PROGRAM MAIN
VAR
	EtapeEnCours:string(50);
END_VAR
VAR // added by the converter: edge detectors and wires of the graphical bodies
    _w1, _w3, _w4, _w5, _w6, _w7, _w8, _w10 : ANY;
    _w2, _w9 : BOOL;
END_VAR

// note: this text did not pass the execution check against the stored diagram
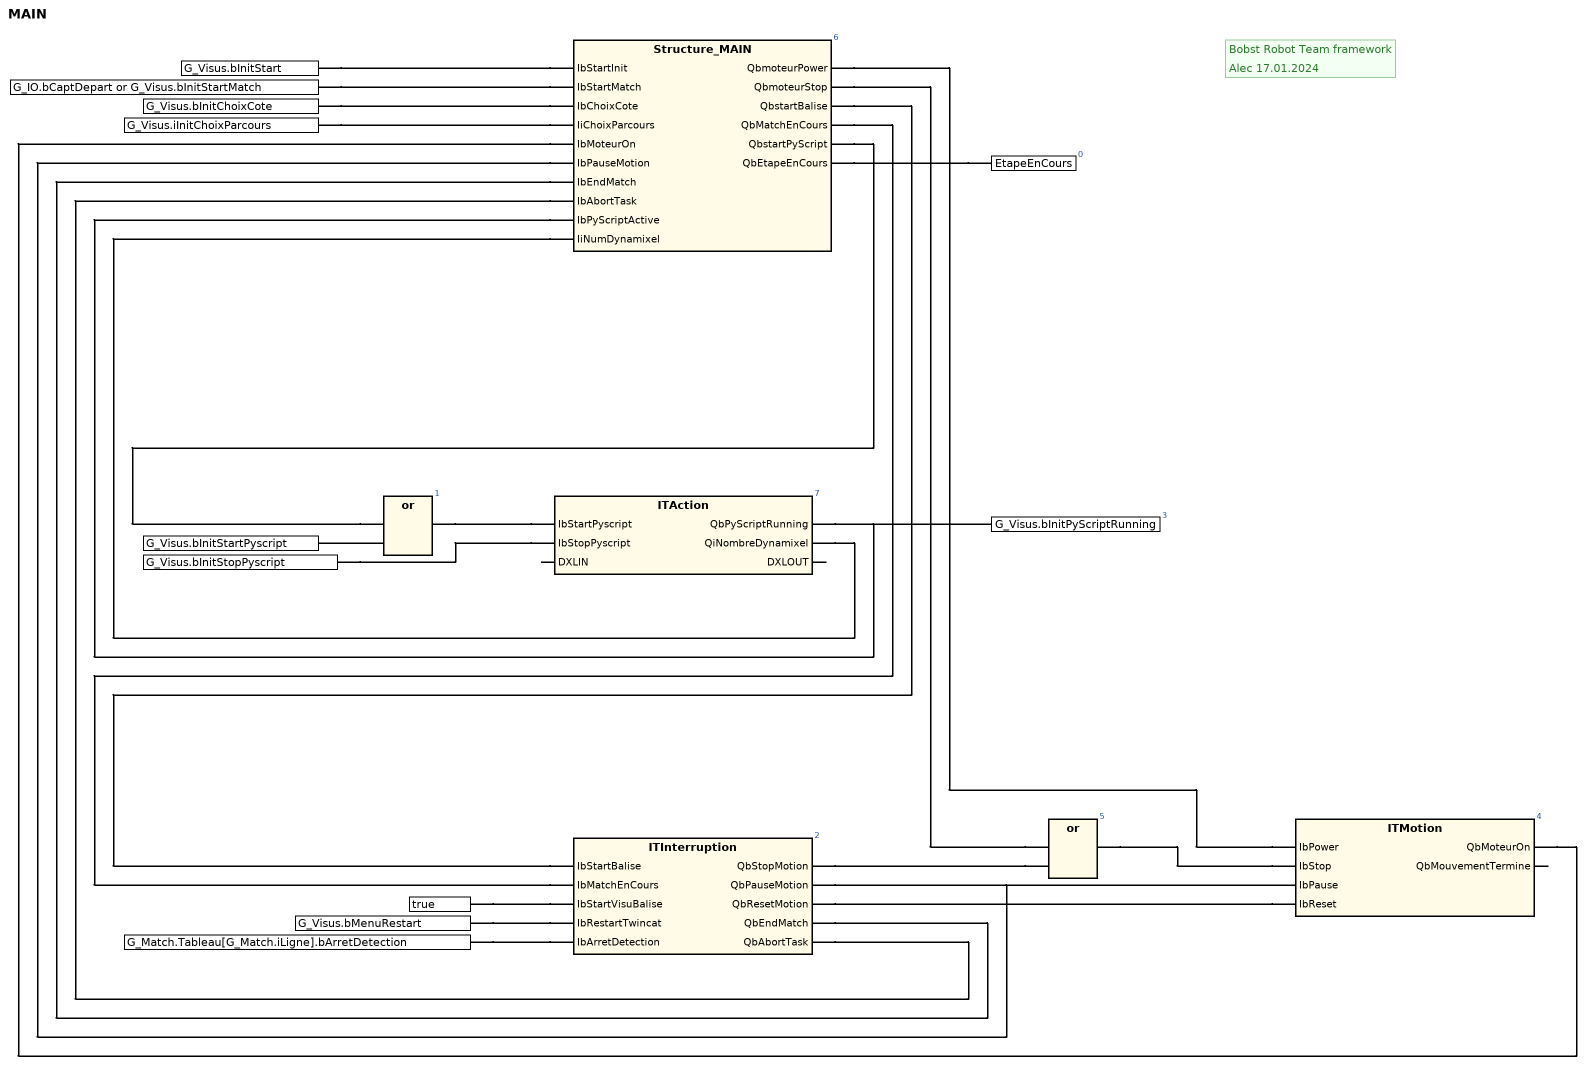
// Bobst Robot Team framework
// Alec 17.01.2024
EtapeEnCours := _w1;
_w3 := _w2 OR G_Visus.bInitStartPyscript;
ITInterruption(IbStartBalise := _w4, IbMatchEnCours := _w5, IbStartVisuBalise := true, IbRestartTwincat := G_Visus.bMenuRestart, IbArretDetection := G_Match.Tableau[G_Match.iLigne].bArretDetection);
G_Visus.bInitPyScriptRunning := _w6;
ITMotion(IbPower := _w7, IbStop := _w8, IbPause := ITInterruption.QbPauseMotion, IbReset := ITInterruption.QbResetMotion);
_w8 := _w9 OR ITInterruption.QbStopMotion;
Structure_MAIN(IbStartInit := G_Visus.bInitStart, IbStartMatch := G_IO.bCaptDepart or G_Visus.bInitStartMatch, IbChoixCote := G_Visus.bInitChoixCote, IiChoixParcours := G_Visus.iInitChoixParcours, IbMoteurOn := ITMotion.QbMoteurOn, IbPauseMotion := ITInterruption.QbPauseMotion, IbEndMatch := ITInterruption.QbEndMatch, IbAbortTask := ITInterruption.QbAbortTask, IbPyScriptActive := _w6, IiNumDynamixel := _w10);
ITAction(IbStartPyscript := _w3, IbStopPyscript := G_Visus.bInitStopPyscript);

END_PROGRAM

(* stored: Version 1.1.0.1, ProductVersion 3.1.4024.12
   POU MAIN: Id {2290ac80-4402-41db-928b-e5eec0cf03b8}, SpecialFunc None *)
